// TIA Portal V17 export
// export: Created 2025-03-07T09:17:29.2924813Z, ExportSetting WithDefaults, DisplayName Totally Integrated Automation Portal, DisplayVersion V17 Update 8, DisplayName TIA Portal Openness, DisplayVersion V17 Update 8, DisplayName TIA Portal Version Control Interface, DisplayVersion V17, DisplayName SINAMICS Startdrive Advanced, DisplayVersion V17 SP2, DisplayName SINAMICS Startdrive G110M, G120, G120C, G120D, G120P, G115D, DisplayVersion V17 SP2, DisplayName SINAMICS Startdrive G130, G150, S120, S150, SINAMICS MV, S210, DisplayVersion V17 SP2, DisplayName STEP 7 Professional, DisplayVersion V17 Update 8, DisplayName SINUMERIK ONE STEP 7 Toolbox, DisplayVersion V17 Update 12, DisplayName SINUMERIK 840D sl STEP 7 Toolbox, DisplayVersion V17 Update 12, DisplayName STEP 7 Safety, DisplayVersion V17 Update 6, DisplayName WinCC Advanced, DisplayVersion V17 Update 8
FUNCTION "FC328_CHANNEL_8" : Void   // FC328, LAD
{ S7_Optimized_Access := 'FALSE' }
AUTHOR : ETXETAR
VERSION : 1.0
// stored: AutoNumber false, IsIECCheckEnabled false, SetENOAutomatically false, UDAEnableTagReadback false
   VAR_TEMP
      NC_RESET_CH4 : Bool;
      NC_START_CH4 : Bool;
   END_VAR
BEGIN

REGION Network 1: RESET CHANNEL
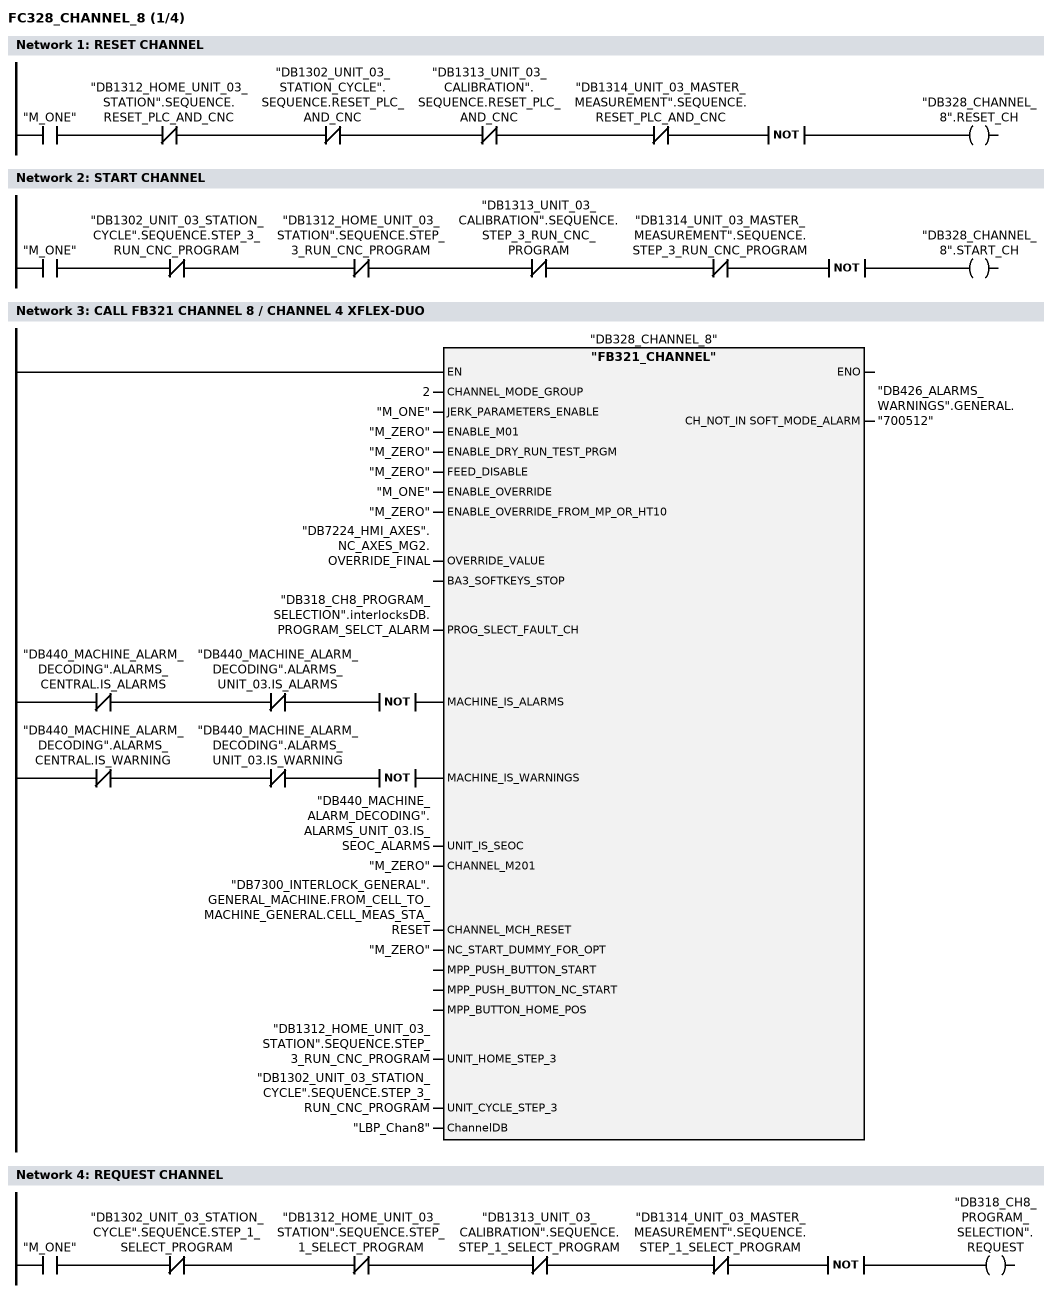
   RUNG wire#powerrail
      Contact( "M_ONE" )
      I_Contact( "DB1312_HOME_UNIT_03_STATION".SEQUENCE.RESET_PLC_AND_CNC )
      I_Contact( "DB1302_UNIT_03_STATION_CYCLE".SEQUENCE.RESET_PLC_AND_CNC )
      I_Contact( "DB1313_UNIT_03_CALIBRATION".SEQUENCE.RESET_PLC_AND_CNC )
      I_Contact( "DB1314_UNIT_03_MASTER_MEASUREMENT".SEQUENCE.RESET_PLC_AND_CNC )
      Not()
      Coil( "DB328_CHANNEL_8".RESET_CH )
   END_RUNG
   // the same network as SCL:
   "DB328_CHANNEL_8".RESET_CH := NOT ("M_ONE" AND NOT "DB1312_HOME_UNIT_03_STATION".SEQUENCE.RESET_PLC_AND_CNC AND NOT "DB1302_UNIT_03_STATION_CYCLE".SEQUENCE.RESET_PLC_AND_CNC AND NOT "DB1313_UNIT_03_CALIBRATION".SEQUENCE.RESET_PLC_AND_CNC AND NOT "DB1314_UNIT_03_MASTER_MEASUREMENT".SEQUENCE.RESET_PLC_AND_CNC);
END_REGION

REGION Network 2: START CHANNEL
   RUNG wire#powerrail
      Contact( "M_ONE" )
      I_Contact( "DB1302_UNIT_03_STATION_CYCLE".SEQUENCE.STEP_3_RUN_CNC_PROGRAM )
      I_Contact( "DB1312_HOME_UNIT_03_STATION".SEQUENCE.STEP_3_RUN_CNC_PROGRAM )
      I_Contact( "DB1313_UNIT_03_CALIBRATION".SEQUENCE.STEP_3_RUN_CNC_PROGRAM )
      I_Contact( "DB1314_UNIT_03_MASTER_MEASUREMENT".SEQUENCE.STEP_3_RUN_CNC_PROGRAM )
      Not()
      Coil( "DB328_CHANNEL_8".START_CH )
   END_RUNG
   // the same network as SCL:
   "DB328_CHANNEL_8".START_CH := NOT ("M_ONE" AND NOT "DB1302_UNIT_03_STATION_CYCLE".SEQUENCE.STEP_3_RUN_CNC_PROGRAM AND NOT "DB1312_HOME_UNIT_03_STATION".SEQUENCE.STEP_3_RUN_CNC_PROGRAM AND NOT "DB1313_UNIT_03_CALIBRATION".SEQUENCE.STEP_3_RUN_CNC_PROGRAM AND NOT "DB1314_UNIT_03_MASTER_MEASUREMENT".SEQUENCE.STEP_3_RUN_CNC_PROGRAM);
END_REGION

REGION Network 3: CALL FB321 CHANNEL 8 / CHANNEL 4 XFLEX-DUO
   RUNG wire#powerrail
      "DB328_CHANNEL_8"(MACHINE_IS_ALARMS := wire#w1, MACHINE_IS_WARNINGS := wire#w2, CHANNEL_MODE_GROUP := 2, JERK_PARAMETERS_ENABLE := "M_ONE", ENABLE_M01 := "M_ZERO", ENABLE_DRY_RUN_TEST_PRGM := "M_ZERO", FEED_DISABLE := "M_ZERO", ENABLE_OVERRIDE := "M_ONE", ENABLE_OVERRIDE_FROM_MP_OR_HT10 := "M_ZERO", OVERRIDE_VALUE := "DB7224_HMI_AXES".NC_AXES_MG2.OVERRIDE_FINAL, BA3_SOFTKEYS_STOP :=, PROG_SLECT_FAULT_CH := "DB318_CH8_PROGRAM_SELECTION".interlocksDB.PROGRAM_SELCT_ALARM, UNIT_IS_SEOC := "DB440_MACHINE_ALARM_DECODING".ALARMS_UNIT_03.IS_SEOC_ALARMS, CHANNEL_M201 := "M_ZERO", CHANNEL_MCH_RESET := "DB7300_INTERLOCK_GENERAL".GENERAL_MACHINE.FROM_CELL_TO_MACHINE_GENERAL.CELL_MEAS_STA_RESET, NC_START_DUMMY_FOR_OPT := "M_ZERO", MPP_PUSH_BUTTON_START :=, MPP_PUSH_BUTTON_NC_START :=, MPP_BUTTON_HOME_POS :=, UNIT_HOME_STEP_3 := "DB1312_HOME_UNIT_03_STATION".SEQUENCE.STEP_3_RUN_CNC_PROGRAM, UNIT_CYCLE_STEP_3 := "DB1302_UNIT_03_STATION_CYCLE".SEQUENCE.STEP_3_RUN_CNC_PROGRAM, ChannelDB := "LBP_Chan8", "CH_NOT_IN SOFT_MODE_ALARM" => "DB426_ALARMS_WARNINGS".GENERAL."700512")
   END_RUNG
   RUNG wire#powerrail
      I_Contact( "DB440_MACHINE_ALARM_DECODING".ALARMS_CENTRAL.IS_ALARMS )
      I_Contact( "DB440_MACHINE_ALARM_DECODING".ALARMS_UNIT_03.IS_ALARMS )
      Not()
   END_RUNG wire#w1
   RUNG wire#powerrail
      I_Contact( "DB440_MACHINE_ALARM_DECODING".ALARMS_CENTRAL.IS_WARNING )
      I_Contact( "DB440_MACHINE_ALARM_DECODING".ALARMS_UNIT_03.IS_WARNING )
      Not()
   END_RUNG wire#w2
   // the same network as SCL:
   "DB328_CHANNEL_8"(CHANNEL_MODE_GROUP := 2,   // "FB321_CHANNEL"
                     JERK_PARAMETERS_ENABLE := "M_ONE",
                     ENABLE_M01 := "M_ZERO",
                     ENABLE_DRY_RUN_TEST_PRGM := "M_ZERO",
                     FEED_DISABLE := "M_ZERO",
                     ENABLE_OVERRIDE := "M_ONE",
                     ENABLE_OVERRIDE_FROM_MP_OR_HT10 := "M_ZERO",
                     OVERRIDE_VALUE := "DB7224_HMI_AXES".NC_AXES_MG2.OVERRIDE_FINAL,
                     PROG_SLECT_FAULT_CH := "DB318_CH8_PROGRAM_SELECTION".interlocksDB.PROGRAM_SELCT_ALARM,
                     MACHINE_IS_ALARMS := NOT (NOT "DB440_MACHINE_ALARM_DECODING".ALARMS_CENTRAL.IS_ALARMS AND NOT "DB440_MACHINE_ALARM_DECODING".ALARMS_UNIT_03.IS_ALARMS),
                     MACHINE_IS_WARNINGS := NOT (NOT "DB440_MACHINE_ALARM_DECODING".ALARMS_CENTRAL.IS_WARNING AND NOT "DB440_MACHINE_ALARM_DECODING".ALARMS_UNIT_03.IS_WARNING),
                     UNIT_IS_SEOC := "DB440_MACHINE_ALARM_DECODING".ALARMS_UNIT_03.IS_SEOC_ALARMS,
                     CHANNEL_M201 := "M_ZERO",
                     CHANNEL_MCH_RESET := "DB7300_INTERLOCK_GENERAL".GENERAL_MACHINE.FROM_CELL_TO_MACHINE_GENERAL.CELL_MEAS_STA_RESET,
                     NC_START_DUMMY_FOR_OPT := "M_ZERO",
                     UNIT_HOME_STEP_3 := "DB1312_HOME_UNIT_03_STATION".SEQUENCE.STEP_3_RUN_CNC_PROGRAM,
                     UNIT_CYCLE_STEP_3 := "DB1302_UNIT_03_STATION_CYCLE".SEQUENCE.STEP_3_RUN_CNC_PROGRAM,
                     ChannelDB := "LBP_Chan8",
                     "CH_NOT_IN SOFT_MODE_ALARM" => "DB426_ALARMS_WARNINGS".GENERAL."700512");
END_REGION

REGION Network 4: REQUEST CHANNEL
   RUNG wire#powerrail
      Contact( "M_ONE" )
      I_Contact( "DB1302_UNIT_03_STATION_CYCLE".SEQUENCE.STEP_1_SELECT_PROGRAM )
      I_Contact( "DB1312_HOME_UNIT_03_STATION".SEQUENCE.STEP_1_SELECT_PROGRAM )
      I_Contact( "DB1313_UNIT_03_CALIBRATION".SEQUENCE.STEP_1_SELECT_PROGRAM )
      I_Contact( "DB1314_UNIT_03_MASTER_MEASUREMENT".SEQUENCE.STEP_1_SELECT_PROGRAM )
      Not()
      Coil( "DB318_CH8_PROGRAM_SELECTION".REQUEST )
   END_RUNG
   // the same network as SCL:
   "DB318_CH8_PROGRAM_SELECTION".REQUEST := NOT ("M_ONE" AND NOT "DB1302_UNIT_03_STATION_CYCLE".SEQUENCE.STEP_1_SELECT_PROGRAM AND NOT "DB1312_HOME_UNIT_03_STATION".SEQUENCE.STEP_1_SELECT_PROGRAM AND NOT "DB1313_UNIT_03_CALIBRATION".SEQUENCE.STEP_1_SELECT_PROGRAM AND NOT "DB1314_UNIT_03_MASTER_MEASUREMENT".SEQUENCE.STEP_1_SELECT_PROGRAM);
END_REGION

REGION Network 5: CALL FB311 CHANNEL PROGRAM SELECTION / CHANNEL 4 X-FLEX DUO
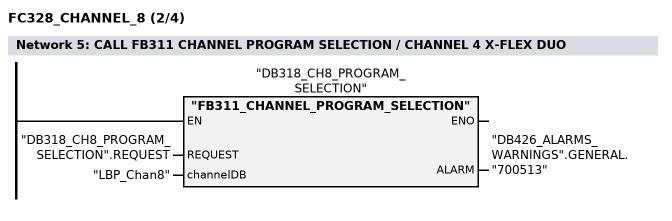
   RUNG wire#powerrail
      "DB318_CH8_PROGRAM_SELECTION"(REQUEST := "DB318_CH8_PROGRAM_SELECTION".REQUEST, channelDB := "LBP_Chan8", ALARM => "DB426_ALARMS_WARNINGS".GENERAL."700513")
   END_RUNG
   // the same network as SCL:
   "DB318_CH8_PROGRAM_SELECTION"(REQUEST := "DB318_CH8_PROGRAM_SELECTION".REQUEST,   // "FB311_CHANNEL_PROGRAM_SELECTION"
                           channelDB := "LBP_Chan8",
                           ALARM => "DB426_ALARMS_WARNINGS".GENERAL."700513");
END_REGION

REGION Network 6: CALL FB301 CHANNEL READ AXES POSITIONS
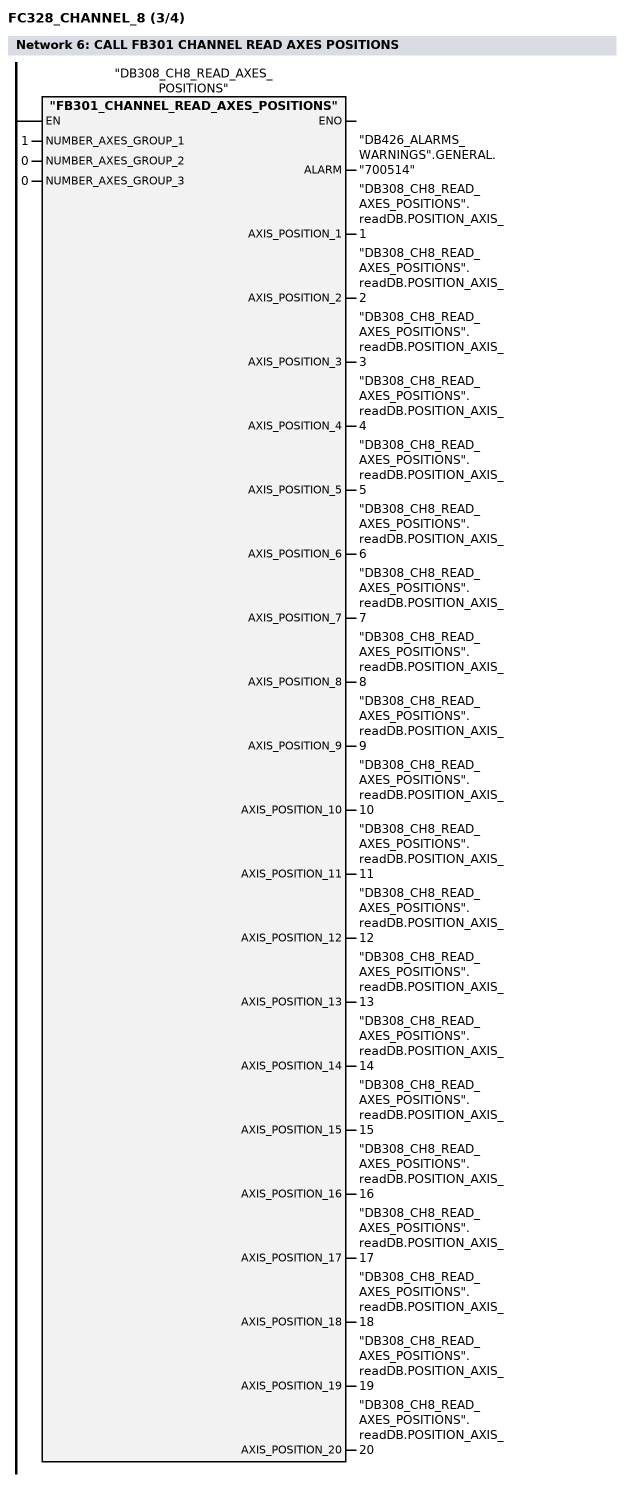
   RUNG wire#powerrail
      "DB308_CH8_READ_AXES_POSITIONS"(NUMBER_AXES_GROUP_1 := 1, NUMBER_AXES_GROUP_2 := 0, NUMBER_AXES_GROUP_3 := 0, ALARM => "DB426_ALARMS_WARNINGS".GENERAL."700514", AXIS_POSITION_1 => "DB308_CH8_READ_AXES_POSITIONS".readDB.POSITION_AXIS_1, AXIS_POSITION_2 => "DB308_CH8_READ_AXES_POSITIONS".readDB.POSITION_AXIS_2, AXIS_POSITION_3 => "DB308_CH8_READ_AXES_POSITIONS".readDB.POSITION_AXIS_3, AXIS_POSITION_4 => "DB308_CH8_READ_AXES_POSITIONS".readDB.POSITION_AXIS_4, AXIS_POSITION_5 => "DB308_CH8_READ_AXES_POSITIONS".readDB.POSITION_AXIS_5, AXIS_POSITION_6 => "DB308_CH8_READ_AXES_POSITIONS".readDB.POSITION_AXIS_6, AXIS_POSITION_7 => "DB308_CH8_READ_AXES_POSITIONS".readDB.POSITION_AXIS_7, AXIS_POSITION_8 => "DB308_CH8_READ_AXES_POSITIONS".readDB.POSITION_AXIS_8, AXIS_POSITION_9 => "DB308_CH8_READ_AXES_POSITIONS".readDB.POSITION_AXIS_9, AXIS_POSITION_10 => "DB308_CH8_READ_AXES_POSITIONS".readDB.POSITION_AXIS_10, AXIS_POSITION_11 => "DB308_CH8_READ_AXES_POSITIONS".readDB.POSITION_AXIS_11, AXIS_POSITION_12 => "DB308_CH8_READ_AXES_POSITIONS".readDB.POSITION_AXIS_12, AXIS_POSITION_13 => "DB308_CH8_READ_AXES_POSITIONS".readDB.POSITION_AXIS_13, AXIS_POSITION_14 => "DB308_CH8_READ_AXES_POSITIONS".readDB.POSITION_AXIS_14, AXIS_POSITION_15 => "DB308_CH8_READ_AXES_POSITIONS".readDB.POSITION_AXIS_15, AXIS_POSITION_16 => "DB308_CH8_READ_AXES_POSITIONS".readDB.POSITION_AXIS_16, AXIS_POSITION_17 => "DB308_CH8_READ_AXES_POSITIONS".readDB.POSITION_AXIS_17, AXIS_POSITION_18 => "DB308_CH8_READ_AXES_POSITIONS".readDB.POSITION_AXIS_18, AXIS_POSITION_19 => "DB308_CH8_READ_AXES_POSITIONS".readDB.POSITION_AXIS_19, AXIS_POSITION_20 => "DB308_CH8_READ_AXES_POSITIONS".readDB.POSITION_AXIS_20)
   END_RUNG
   // the same network as SCL:
   "DB308_CH8_READ_AXES_POSITIONS"(NUMBER_AXES_GROUP_1 := 1,   // "FB301_CHANNEL_READ_AXES_POSITIONS"
                           NUMBER_AXES_GROUP_2 := 0,
                           NUMBER_AXES_GROUP_3 := 0,
                           ALARM => "DB426_ALARMS_WARNINGS".GENERAL."700514",
                           AXIS_POSITION_1 => "DB308_CH8_READ_AXES_POSITIONS".readDB.POSITION_AXIS_1,
                           AXIS_POSITION_2 => "DB308_CH8_READ_AXES_POSITIONS".readDB.POSITION_AXIS_2,
                           AXIS_POSITION_3 => "DB308_CH8_READ_AXES_POSITIONS".readDB.POSITION_AXIS_3,
                           AXIS_POSITION_4 => "DB308_CH8_READ_AXES_POSITIONS".readDB.POSITION_AXIS_4,
                           AXIS_POSITION_5 => "DB308_CH8_READ_AXES_POSITIONS".readDB.POSITION_AXIS_5,
                           AXIS_POSITION_6 => "DB308_CH8_READ_AXES_POSITIONS".readDB.POSITION_AXIS_6,
                           AXIS_POSITION_7 => "DB308_CH8_READ_AXES_POSITIONS".readDB.POSITION_AXIS_7,
                           AXIS_POSITION_8 => "DB308_CH8_READ_AXES_POSITIONS".readDB.POSITION_AXIS_8,
                           AXIS_POSITION_9 => "DB308_CH8_READ_AXES_POSITIONS".readDB.POSITION_AXIS_9,
                           AXIS_POSITION_10 => "DB308_CH8_READ_AXES_POSITIONS".readDB.POSITION_AXIS_10,
                           AXIS_POSITION_11 => "DB308_CH8_READ_AXES_POSITIONS".readDB.POSITION_AXIS_11,
                           AXIS_POSITION_12 => "DB308_CH8_READ_AXES_POSITIONS".readDB.POSITION_AXIS_12,
                           AXIS_POSITION_13 => "DB308_CH8_READ_AXES_POSITIONS".readDB.POSITION_AXIS_13,
                           AXIS_POSITION_14 => "DB308_CH8_READ_AXES_POSITIONS".readDB.POSITION_AXIS_14,
                           AXIS_POSITION_15 => "DB308_CH8_READ_AXES_POSITIONS".readDB.POSITION_AXIS_15,
                           AXIS_POSITION_16 => "DB308_CH8_READ_AXES_POSITIONS".readDB.POSITION_AXIS_16,
                           AXIS_POSITION_17 => "DB308_CH8_READ_AXES_POSITIONS".readDB.POSITION_AXIS_17,
                           AXIS_POSITION_18 => "DB308_CH8_READ_AXES_POSITIONS".readDB.POSITION_AXIS_18,
                           AXIS_POSITION_19 => "DB308_CH8_READ_AXES_POSITIONS".readDB.POSITION_AXIS_19,
                           AXIS_POSITION_20 => "DB308_CH8_READ_AXES_POSITIONS".readDB.POSITION_AXIS_20);
END_REGION

REGION Network 7: CALL FC353 NCK M UNIT 03 / CALL FC1182
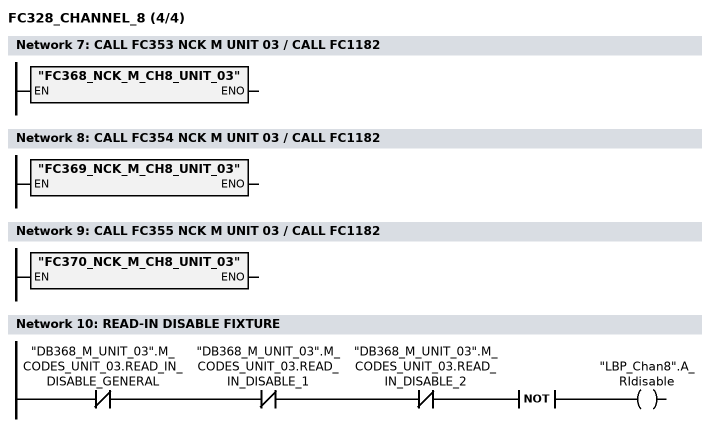
   RUNG wire#powerrail
      "FC368_NCK_M_CH8_UNIT_03"()
   END_RUNG
   // the same network as SCL:
   "FC368_NCK_M_CH8_UNIT_03"();
END_REGION

REGION Network 8: CALL FC354 NCK M UNIT 03 / CALL FC1182
   RUNG wire#powerrail
      "FC369_NCK_M_CH8_UNIT_03"()
   END_RUNG
   // the same network as SCL:
   "FC369_NCK_M_CH8_UNIT_03"();
END_REGION

REGION Network 9: CALL FC355 NCK M UNIT 03 / CALL FC1182
   RUNG wire#powerrail
      "FC370_NCK_M_CH8_UNIT_03"()
   END_RUNG
   // the same network as SCL:
   "FC370_NCK_M_CH8_UNIT_03"();
END_REGION

REGION Network 10: READ-IN DISABLE FIXTURE
   RUNG wire#powerrail
      I_Contact( "DB368_M_UNIT_03".M_CODES_UNIT_03.READ_IN_DISABLE_GENERAL )
      I_Contact( "DB368_M_UNIT_03".M_CODES_UNIT_03.READ_IN_DISABLE_1 )
      I_Contact( "DB368_M_UNIT_03".M_CODES_UNIT_03.READ_IN_DISABLE_2 )
      Not()
      Coil( "LBP_Chan8".A_RIdisable )
   END_RUNG
   // the same network as SCL:
   "LBP_Chan8".A_RIdisable := NOT (NOT "DB368_M_UNIT_03".M_CODES_UNIT_03.READ_IN_DISABLE_GENERAL AND NOT "DB368_M_UNIT_03".M_CODES_UNIT_03.READ_IN_DISABLE_1 AND NOT "DB368_M_UNIT_03".M_CODES_UNIT_03.READ_IN_DISABLE_2);
END_REGION
END_FUNCTION
